(* CoDeSys 2.3.9.25 project: Slunce_vypocet_pohybu_po_obloze_SUNSET.pro *)
(* Libraries: Building_common.lib 26.8.08 09:44:32, SysLibTime.lib 5.10.04 10:39:34, D:\_WAGO\IO_Pro_CAA\library\DaylightSaving.lib 22.2.07 11:46:44, SysLibRtc.lib 5.10.04 10:37:42, D:\_WAGO\IO_Pro_CAA\library\WagoLibDaylightSaving.lib 19.9.06 14:57:10, Standard.lib 22.11.04 11:21:12, SYSLIBCALLBACK.LIB 20.4.05 11:04:48 *)

(* PLC configuration (modules and I/O channels)
K-Bus [K_Bus] node 0, in %IB0 out %QB0
  0750-0502 2 DO 24V DC 2.0A [Type_10_2_Channels] node 0, in %IB0 out %QB0 {INTTypePAAssignment = PLC; INTTypeModule = plugged}
    AT %QX4.0 [BOOLOnX_Q] Ch_1 Digital output
    AT %QX4.1 [BOOLOnX_Q] Ch_2 Digital output
  0750-0530 8 DO 24 V DC 0.5A [Type_10_8_Channels] node 1, in %IB1 out %QB1 {INTTypePAAssignment = PLC; INTTypeModule = plugged}
    AT %QX4.2 [BOOLOnX_Q] Ch_1 Digital output
    AT %QX4.3 [BOOLOnX_Q] Ch_2 Digital output
    AT %QX4.4 [BOOLOnX_Q] Ch_3 Digital output
    AT %QX4.5 [BOOLOnX_Q] Ch_4 Digital output
    AT %QX4.6 [BOOLOnX_Q] Ch_5 Digital output
    AT %QX4.7 [BOOLOnX_Q] Ch_6 Digital output
    AT %QX4.8 [BOOLOnX_Q] Ch_7 Digital output
    AT %QX4.9 [BOOLOnX_Q] Ch_8 Digital output
  0750-0430 8 DI 24 V DC 3.0ms [Type_1_8_Channels] node 3, in %IB3 out %QB3 {INTTypePAAssignment = PLC; INTTypeModule = plugged}
    AT %IX6.0 [BOOLOnX_I] Ch_1 Digital input
    AT %IX6.1 [BOOLOnX_I] Ch_2 Digital input
    AT %IX6.2 [BOOLOnX_I] Ch_3 Digital input
    AT %IX6.3 [BOOLOnX_I] Ch_4 Digital input
    AT %IX6.4 [BOOLOnX_I] Ch_5 Digital input
    AT %IX6.5 [BOOLOnX_I] Ch_6 Digital input
    AT %IX6.6 [BOOLOnX_I] Ch_7 Digital input
    AT %IX6.7 [BOOLOnX_I] Ch_8 Digital input
  0750-0430 8 DI 24 V DC 3.0ms [Type_1_8_Channels] node 4, in %IB4 out %QB4 {INTTypePAAssignment = PLC; INTTypeModule = plugged}
    AT %IX6.8 [BOOLOnX_I] Ch_1 Digital input
    AT %IX6.9 [BOOLOnX_I] Ch_2 Digital input
    AT %IX6.10 [BOOLOnX_I] Ch_3 Digital input
    AT %IX6.11 [BOOLOnX_I] Ch_4 Digital input
    AT %IX6.12 [BOOLOnX_I] Ch_5 Digital input
    AT %IX6.13 [BOOLOnX_I] Ch_6 Digital input
    AT %IX6.14 [BOOLOnX_I] Ch_7 Digital input
    AT %IX6.15 [BOOLOnX_I] Ch_8 Digital input
  0750-0464#02 2/4 AI RTD / ADJ./ HA [Type_44_2_Channels] node 5, in %IB5 out %QB5 {INTTypePAAssignment = PLC; INTTypeModule = plugged}
    AT %IW0 [INTOnW_I] Ch_1 signed Input value
    AT %IW1 [INTOnW_I] Ch_2 signed Input value
  0750-0559 4 AO 0-10V DC [Type_14_4_Channels] node 6, in %IB6 out %QB6 {INTTypePAAssignment = PLC; INTTypeModule = plugged}
    AT %QW0 [WORDOnW_Q] Ch_1 Analog output
    AT %QW1 [WORDOnW_Q] Ch_2 Analog output
    AT %QW2 [WORDOnW_Q] Ch_3 Analog output
    AT %QW3 [WORDOnW_Q] Ch_4 Analog output
  0750-0455 4 AI 4-20mA s.e. [Type_8_4_Channels] node 7, in %IB7 out %QB7 {INTTypePAAssignment = PLC; INTTypeModule = plugged}
    AT %IW2 [WORDOnW_I] Ch_1 Input word
    AT %IW3 [WORDOnW_I] Ch_2 Input word
    AT %IW4 [WORDOnW_I] Ch_3 Input word
    AT %IW5 [WORDOnW_I] Ch_4 Input word
Fieldbus variables [FB_VARS] node 1, in %IB0 out %QB0
*)

(* Task configuration *)
TASK slunce (PRIORITY := 15, INTERVAL := T#1000ms);
	Vypocet_pohybu_slunce();
END_TASK

(* POU Vypocet_pohybu_slunce, CFC *)
PROGRAM Vypocet_pohybu_slunce
(*Program vypocte pohyb slunce po obloze na zaklade aktualnicho data a casu v systemu,
Zemepisna sirka/delka jsou nastavena na Prahu, lze libovolne zmenit.
Vystupnimi hodnotami jsou Azimut a Elevace. Pokud je Elevace<0 - Slunce zapadlo.
Vytvoreno pro procesory s 32 bitovou architekturou.
Program se spousti kazdou 1 s, jako cyklický task.
Testovano na 750-841, 750-873 	
2009-07-13 Ondrej Dolejs*)

VAR
	Pohyb_slunce: Fb_Sunset;
	AktualniCas: DT;
	UTCiCas: DT;		(*Odpovídá casu GMT, rozdíl pouze v rozsahu [s]*)
	ZemepisnaSirka: 	REAL := 50.083333333;		(*Praha 50 stupnu a 5 minut N, prepocteno stupne + minuty/60*)
	ZemepisnaDelka: REAL := 14.433333333;		(*Praha 14 stupnu a 26 minut E, prepocteno stupne + minuty/60*)
	Elevace: REAL;		(*uhel slunce nad obzorem*)
	Azimut: REAL;			(*Sever 0 stupnu, jih 180 stupnu*)
	leto: BOOL;			(*TRUE, když je leto*)
	DenVtydnu: BYTE;		(*Pondeli=1, utery=2,...., nedele=7*)
END_VAR
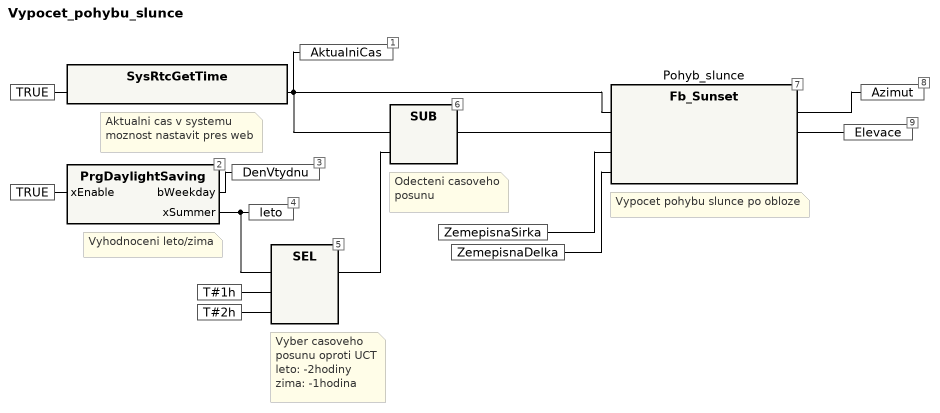
_CFC_ (* Continuous Function Chart, elements in execution order *)
#0 SysRtcGetTime(TRUE)
(* Vyber casoveho / posunu oproti UCT / leto: -2hodiny / zima: -1hodina *)
(* Aktualni cas v systemu / moznost nastavit pres web *)
(* Odecteni casoveho / posunu *)
(* Vypocet pohybu slunce po obloze *)
#1 AktualniCas <= #0
#2 PrgDaylightSaving(xEnable: TRUE)
#3 DenVtydnu <= #2.bWeekday
#4 leto <= #2.xSummer
#5 SEL(#2.xSummer, T#1h, T#2h)
#6 SUB(#0, #5)
#7 Pohyb_slunce:Fb_Sunset(#0, #6, ZemepisnaSirka, ZemepisnaDelka)
#8 Azimut <= #7.out 1
#9 Elevace <= #7.out 2
(* Vyhodnoceni leto/zima *)
_END_CFC_
END_PROGRAM
